Staubli VAL3: interfaceCS9.pjx

--- interfaceCS9.pjx ---
Parameters version=s7.11 stackSize=5000 millimeterUnit=true
Program file=ack.pgx
Program file=clearScreen.pgx
Program file=debug.pgx
Program file=feedbackStatus.pgx
Program file=init.pgx
Program file=motionBuffer.pgx
Program file=motionProgress.pgx
Program file=motionStatus.pgx
Program file=start.pgx
Program file=stop.pgx
Program file=trajBuffer.pgx
Program file=velOverwrite.pgx
Data file=interfaceCS9.dtx
Library alias=libQueueFuncs path=Disk://ros_libs/QueueFuncs/QueueFuncs.pjx

--- interfaceCS9.dtx ---
mdesc mNomSpeed

--- start.pgx ---
program start()
begin

  // Library to handle all of the interface actions for CS9 controller
  // Loaded at runtime in ros_server()

  // DO NOT auto-load
  // Auto-loading will break cross-controller functionality
  // The correct library will be loaded at runtime, otherwise an error will be generated

end

--- ack.pgx ---
public program ack(num x_nHeaderTime, num x_nElapsedTime)
begin

  // display time between valid trajectory point received and ACK sent
  userPageSet("uxMonitor", "lblHeaderTime", "innerHTML", toString(".4", x_nHeaderTime))
  userPageSet("uxMonitor", "lblElapsedTime", "innerHTML", toString(".4", x_nElapsedTime))

end

--- clearScreen.pgx ---
public program clearScreen()
begin

  // Do nothing - not needed on CS9

end

--- debug.pgx ---
public program debug(num& x_nExecStatus)
begin

  // Do nothing - not needed on CS9

end

--- feedbackStatus.pgx ---
public program feedbackStatus(num x_nOutConnFlag)
begin

  // update connection status on port 11002
  switch x_nOutConnFlag
    case -1
      userPageSet("uxMonitor", "lblFeedbackState", "innerHTML", "connection lost")
    break
    case 0
      userPageSet("uxMonitor", "lblFeedbackState", "innerHTML", "not connected")
    break
    case 1
      userPageSet("uxMonitor", "lblFeedbackState", "innerHTML", "connected")
    break
    default
      userPageSet("uxMonitor", "lblFeedbackState", "innerHTML", "not connected")
    break
  endSwitch

end

--- init.pgx ---
public program init()
begin


  userPage("uxMonitor")

end

--- motionBuffer.pgx ---
public program motionBuffer(num x_nMovePts, num x_nElems)
begin

  userPageSet("uxMonitor", "lblMotionBuffer", "innerHTML", x_nElems)
  userPageSet("uxMonitor", "lblMotionBufferPopped", "innerHTML", x_nMovePts)

end

--- motionProgress.pgx ---
public program motionProgress(num x_nMoveId, num x_nMotProg)
begin

  // display nMoveId and nMotionProgress
  userPageSet("uxMonitor", "lblMoveId", "innerHTML", x_nMoveId)
  userPageSet("uxMonitor", "lblMotionProgress", "innerHTML", x_nMotProg)

end

--- motionStatus.pgx ---
public program motionStatus(num x_nInConnFlag)
begin

  // update connection status on port 11000
    switch x_nInConnFlag
      case -1
        userPageSet("uxMonitor", "lblMotionState", "innerHTML", "connection lost")
      break
      case 0
        userPageSet("uxMonitor", "lblMotionState", "innerHTML", "not connected")
      break
      case 1
        userPageSet("uxMonitor", "lblMotionState", "innerHTML", "connected")
      break
      default
        userPageSet("uxMonitor", "lblMotionState", "innerHTML", "not connected")
      break
    endSwitch

end

--- trajBuffer.pgx ---
public program trajBuffer(num x_nElems, num x_nPtsPopped)
begin

  userPageSet("uxMonitor", "lblTrajectoryBuffer", "innerHTML", x_nElems)
  userPageSet("uxMonitor", "lblTrajectoryBufferPopped", "innerHTML", x_nPtsPopped)

end

--- velOverwrite.pgx ---
public program velOverwrite(bool x_bOverwriteVel)
begin

  // display velocity overwrite status
    if(x_bOverwriteVel == true)
      userPageSet("uxMonitor", "lblVelocityOverwrite", "innerHTML", "enabled")
    else
      userPageSet("uxMonitor", "lblVelocityOverwrite", "innerHTML", "disabled")
    endIf

end
